// TwinCAT 3 PLC project Traffic
// ProgramVersion: 3.1.4024.0
// libraries:
//   Tc2_Standard, * (Beckhoff Automation GmbH)
//   Tc2_System, * (Beckhoff Automation GmbH)
//   Tc3_Module, * (Beckhoff Automation GmbH)
// project tree:
//   DUTs/ ST_ADJLIST.TcDUT, ST_ADJNODE.TcDUT, ST_GRAPH.TcDUT
//   GVLs/ CONSTANTS.TcGVL, GLOBALS.TcGVL
//   / PlcTask.TcTTO
//   POUs/ GET_MIN_DISTANCE_NODE.TcPOU, GET_SHORTEST_PATH.TcPOU, MAIN.TcPOU, DIJKSTRA.TcPOU, SIM_VALUES_CALC.TcPOU, TICK.TcPOU
// real-time tasks:
//   TASK PlcTask: cycle T#10ms, priority 20, ADS port 350

CONFIGURATION Traffic
    RESOURCE PLC ON TwinCAT3
        TASK PlcTask(INTERVAL := T#10ms, PRIORITY := 20);
        PROGRAM MAIN WITH PlcTask : MAIN;
    END_RESOURCE
END_CONFIGURATION

// ---- DUTs/ST_ADJLIST.TcDUT
TYPE ST_ADJLIST :
STRUCT
	aAdjNodes : ARRAY[1..3] OF POINTER TO ST_ADJNODE;
END_STRUCT
END_TYPE

// ---- DUTs/ST_ADJNODE.TcDUT
TYPE ST_ADJNODE :
STRUCT
	nNode	: INT;
	nWeight	: POINTER TO INT;
END_STRUCT
END_TYPE

// ---- DUTs/ST_GRAPH.TcDUT
TYPE ST_GRAPH :
STRUCT
	aAdjLists : ARRAY[1..24] OF POINTER TO ST_ADJLIST;
END_STRUCT
END_TYPE

// ---- GVLs/CONSTANTS.TcGVL
{attribute 'qualified_only'}
VAR_GLOBAL
	nIntMax : INT := 32767;
	
	// Base time in seconds required for <5 cars to pass through a crossroads.
	nBaseWeightSR : INT := 10;
	nBaseWeightL : INT := 20;
	
	// Most significant points in a made-up graph illustrating the intensity of traffic flow at specified hours.
	// aTrafficFlowTimes - X axis
	// aTrafficFlowVals - Y axis
	// To find the value of flow intensity inbetween these points, the following formula is used:
	// if (x2 < x1) x2 := x2 + 24; y := (x - x1) * (y2 - y1) / (x2 - x1) + y1;
	aTrafficFlowTimes : ARRAY[1..4] OF TOD := [TOD#4:0:0, TOD#9:0:0, TOD#12:0:0, TOD#17:0:0];
	aTrafficFlowVals : ARRAY[1..4] OF REAL := [0.0,       1.0,       0.5,        0.9];
	
	// Each day of the week has a different modifier for traffic intensity as well. 1 means Monday, 7 means Sunday.
	aTrafficFlowDaysVals : ARRAY[1..7] OF REAL := [1.0, 0.95, 0.9, 0.85, 0.8, 0.75, 0.7];
	
END_VAR

// ---- GVLs/GLOBALS.TcGVL
{attribute 'qualified_only'}
VAR_GLOBAL

// Settings for all crossroads.
// They indicate what number of cars should pass through specified parts of them when the modifier is 1.0.
// For example, setting nAHxSR to 100 on Mondays should result in 90 cars passing through at 17:00 and only 10 at 4:00.
// x - horizontal part
// y - vertical part
// SR - straights and rights
// L - lefts
nAHxSR, nAHySR, nAHxL, nAHyL : INT;
nBCxSR, nBCySR, nBCxL, nBCyL : INT;
nDExSR, nDEySR, nDExL, nDEyL : INT;
nFGxSR, nFGySR, nFGxL, nFGyL : INT;

// Depending on the time of day and day of week, this modifier will change from 0.0 for when there is no traffic to 1.0 at rush hours.
rModifier : REAL;

// Weights are the final product of nBaseWeightXX + nBaseWeightXX * {setting} / 5 * nModifier
// This is the time in seconds required to pass through a node.
nWeightAHxSR : INT;
nWeightAHySR : INT;
nWeightAHxL  : INT;
nWeightAHyL  : INT;

nWeightBCxSR : INT;
nWeightBCySR : INT;
nWeightBCxL  : INT;
nWeightBCyL  : INT;

nWeightDExSR : INT;
nWeightDEySR : INT;
nWeightDExL  : INT;
nWeightDEyL  : INT;

nWeightFGxSR : INT;
nWeightFGySR : INT;
nWeightFGxL  : INT;
nWeightFGyL  : INT;

// Adjacent nodes in adjacency lists. For example, stNode1to16 indicates the time required to get from node 1 to its adjacent node 16.
// ----- RIGHTS -----
//RIGHTS AH
stNode1to16  : ST_ADJNODE := (nNode:=16, nWeight:=ADR(nWeightAHySR));
stNode17to2  : ST_ADJNODE := (nNode:=2,  nWeight:=ADR(nWeightAHxSR));
stNode23to18 : ST_ADJNODE := (nNode:=18, nWeight:=ADR(nWeightAHySR));
stNode15to24 : ST_ADJNODE := (nNode:=24, nWeight:=ADR(nWeightAHxSR));
//RIGHTS BC
stNode3to17  : ST_ADJNODE := (nNode:=17, nWeight:=ADR(nWeightBCySR));
stNode5to4   : ST_ADJNODE := (nNode:=4,  nWeight:=ADR(nWeightBCxSR));
stNode20to6  : ST_ADJNODE := (nNode:=6,  nWeight:=ADR(nWeightBCySR));
stNode18to19 : ST_ADJNODE := (nNode:=19, nWeight:=ADR(nWeightBCxSR));
//RIGHTS DE
stNode19to21 : ST_ADJNODE := (nNode:=21, nWeight:=ADR(nWeightDEySR));
stNode7to20  : ST_ADJNODE := (nNode:=20, nWeight:=ADR(nWeightDExSR));
stNode9to8   : ST_ADJNODE := (nNode:=8,  nWeight:=ADR(nWeightDEySR));
stNode22to10 : ST_ADJNODE := (nNode:=10, nWeight:=ADR(nWeightDExSR));
//RIGHTS FG
stNode24to14 : ST_ADJNODE := (nNode:=14, nWeight:=ADR(nWeightFGySR));
stNode21to23 : ST_ADJNODE := (nNode:=23, nWeight:=ADR(nWeightFGxSR));
stNode11to22 : ST_ADJNODE := (nNode:=22, nWeight:=ADR(nWeightFGySR));
stNode13to12 : ST_ADJNODE := (nNode:=12, nWeight:=ADR(nWeightFGxSR));
// ----- STRAIGHTS -----
//STRAIGHTS AH
stNode1to24  : ST_ADJNODE := (nNode:=24, nWeight:=ADR(nWeightAHySR));
stNode23to2  : ST_ADJNODE := (nNode:=2,  nWeight:=ADR(nWeightAHySR));
stNode17to16 : ST_ADJNODE := (nNode:=16, nWeight:=ADR(nWeightAHxSR));
stNode15to18 : ST_ADJNODE := (nNode:=18, nWeight:=ADR(nWeightAHxSR));
//STRAIGHTS BC
stNode3to19 : ST_ADJNODE := (nNode:=19, nWeight:=ADR(nWeightBCySR));
stNode20to4 : ST_ADJNODE := (nNode:=4,  nWeight:=ADR(nWeightBCySR));
stNode5to17 : ST_ADJNODE := (nNode:=17, nWeight:=ADR(nWeightBCxSR));
stNode18to6 : ST_ADJNODE := (nNode:=6,  nWeight:=ADR(nWeightBCxSR));
//STRAIGHTS DE
stNode19to10 : ST_ADJNODE := (nNode:=10, nWeight:=ADR(nWeightDEySR));
stNode9to20  : ST_ADJNODE := (nNode:=20, nWeight:=ADR(nWeightDEySR));
stNode7to21  : ST_ADJNODE := (nNode:=21, nWeight:=ADR(nWeightDExSR));
stNode22to8  : ST_ADJNODE := (nNode:=8,  nWeight:=ADR(nWeightDExSR));
//STRAIGHTS FG
stNode24to12 : ST_ADJNODE := (nNode:=12, nWeight:=ADR(nWeightFGySR));
stNode11to23 : ST_ADJNODE := (nNode:=23, nWeight:=ADR(nWeightFGySR));
stNode21to14 : ST_ADJNODE := (nNode:=14, nWeight:=ADR(nWeightFGxSR));
stNode13to22 : ST_ADJNODE := (nNode:=22, nWeight:=ADR(nWeightFGxSR));
// ----- LEFTS -----
//LEFTS AH
stNode1to18  : ST_ADJNODE := (nNode:=18, nWeight:=ADR(nWeightAHyL));
stNode15to2  : ST_ADJNODE := (nNode:=2,  nWeight:=ADR(nWeightAHxL));
stNode17to24 : ST_ADJNODE := (nNode:=24, nWeight:=ADR(nWeightAHxL));
stNode23to16 : ST_ADJNODE := (nNode:=16, nWeight:=ADR(nWeightAHyL));
//LEFTS BC
stNode3to6   : ST_ADJNODE := (nNode:=6,  nWeight:=ADR(nWeightBCyL));
stNode18to4  : ST_ADJNODE := (nNode:=4,  nWeight:=ADR(nWeightBCxL));
stNode5to19  : ST_ADJNODE := (nNode:=19, nWeight:=ADR(nWeightBCxL));
stNode20to17 : ST_ADJNODE := (nNode:=17, nWeight:=ADR(nWeightBCyL));
//LEFTS DE
stNode19to8  : ST_ADJNODE := (nNode:=8,  nWeight:=ADR(nWeightDEyL));
stNode22to20 : ST_ADJNODE := (nNode:=20, nWeight:=ADR(nWeightDExL));
stNode7to10  : ST_ADJNODE := (nNode:=10, nWeight:=ADR(nWeightDExL));
stNode9to21  : ST_ADJNODE := (nNode:=21, nWeight:=ADR(nWeightDEyL));
//LEFTS FG
stNode24to22 : ST_ADJNODE := (nNode:=22, nWeight:=ADR(nWeightFGyL));
stNode13to23 : ST_ADJNODE := (nNode:=23, nWeight:=ADR(nWeightFGxL));
stNode21to12 : ST_ADJNODE := (nNode:=12, nWeight:=ADR(nWeightFGxL));
stNode11to14 : ST_ADJNODE := (nNode:=14, nWeight:=ADR(nWeightFGyL));

// Adjacency lists for all nodes that can act as sources. Note that there are no lists for destination-only nodes,
// namely nodes 2, 4, 6, 8, 10, 12, 14, 16.
stNodesFrom1  : ST_ADJLIST := (aAdjNodes:=[ADR(stNode1to16),  ADR(stNode1to18),  ADR(stNode1to24)]);
stNodesFrom3  : ST_ADJLIST := (aAdjNodes:=[ADR(stNode3to17),  ADR(stNode3to19),  ADR(stNode3to6)]);
stNodesFrom5  : ST_ADJLIST := (aAdjNodes:=[ADR(stNode5to17),  ADR(stNode5to19),  ADR(stNode5to4)]);
stNodesFrom7  : ST_ADJLIST := (aAdjNodes:=[ADR(stNode7to10),  ADR(stNode7to20),  ADR(stNode7to21)]);
stNodesFrom9  : ST_ADJLIST := (aAdjNodes:=[ADR(stNode9to20),  ADR(stNode9to21),  ADR(stNode9to8)]);
stNodesFrom11 : ST_ADJLIST := (aAdjNodes:=[ADR(stNode11to14), ADR(stNode11to22), ADR(stNode11to23)]);
stNodesFrom13 : ST_ADJLIST := (aAdjNodes:=[ADR(stNode13to12), ADR(stNode13to22), ADR(stNode13to23)]);
stNodesFrom15 : ST_ADJLIST := (aAdjNodes:=[ADR(stNode15to18), ADR(stNode15to2),  ADR(stNode15to24)]);
stNodesFrom17 : ST_ADJLIST := (aAdjNodes:=[ADR(stNode17to16), ADR(stNode17to2),  ADR(stNode17to24)]);
stNodesFrom18 : ST_ADJLIST := (aAdjNodes:=[ADR(stNode18to19), ADR(stNode18to4),  ADR(stNode18to6)]);
stNodesFrom19 : ST_ADJLIST := (aAdjNodes:=[ADR(stNode19to10), ADR(stNode19to21), ADR(stNode19to8)]);
stNodesFrom20 : ST_ADJLIST := (aAdjNodes:=[ADR(stNode20to17), ADR(stNode20to4),  ADR(stNode20to6)]);
stNodesFrom21 : ST_ADJLIST := (aAdjNodes:=[ADR(stNode21to12), ADR(stNode21to14), ADR(stNode21to23)]);
stNodesFrom22 : ST_ADJLIST := (aAdjNodes:=[ADR(stNode22to10), ADR(stNode22to20), ADR(stNode22to8)]);
stNodesFrom23 : ST_ADJLIST := (aAdjNodes:=[ADR(stNode23to16), ADR(stNode23to18), ADR(stNode23to2)]);
stNodesFrom24 : ST_ADJLIST := (aAdjNodes:=[ADR(stNode24to12), ADR(stNode24to14), ADR(stNode24to22)]);

// Adjacency graph. Note that destination-only nodes have no adjacency lists; their address is set to 0 and is ignored when searching.
stGraph : ST_GRAPH := (aAdjLists:=[
ADR(stNodesFrom1),
0,
ADR(stNodesFrom3),
0,
ADR(stNodesFrom5),
0,
ADR(stNodesFrom7),
0,
ADR(stNodesFrom9),
0,
ADR(stNodesFrom11),
0,
ADR(stNodesFrom13),
0,
ADR(stNodesFrom15),
0,
ADR(stNodesFrom17),
ADR(stNodesFrom18),
ADR(stNodesFrom19),
ADR(stNodesFrom20),
ADR(stNodesFrom21),
ADR(stNodesFrom22),
ADR(stNodesFrom23),
ADR(stNodesFrom24)]);

// Nodes for the Dijkstra algorithm search.
nStartPosition : INT := 1;
nEndPosition: INT := 2;

// List of all distances from nStartPosition
aDistances : ARRAY[1..24] OF INT;

// List of traveled nodes from nStartPosition to nEndPosition
aRoadFlags : ARRAY[1..24] OF BOOL;

END_VAR

// ---- POUs/MAIN.TcPOU
PROGRAM MAIN
VAR
	bShouldCalculate : BOOL;
END_VAR

TICK();
SIM_VALUES_CALC();
IF bShouldCalculate THEN
	DIJKSTRA();
	bShouldCalculate := FALSE;
END_IF

END_PROGRAM

// ---- POUs/TICK.TcPOU
PROGRAM TICK
VAR
	ins : BOOL;
	et : TIME;
	tick: TON;
	
	nDayOfTheWeek : INT := 1;
	
	tdSimTime : TOD := TOD#4:0:0;
	SimTime : UDINT;
	
	// Traffic flow time index for CONSTANTS.aTrafficFlowTimes
	x1i : INT := 1;
	x2i : INT := 2;
	x1, x2 : REAL;
	
	tdTickTime : TOD := TOD#0:15:0;
END_VAR
VAR // added by the converter: edge detectors and wires of the graphical bodies
    _w1, _w2, _w3 : BOOL;
END_VAR

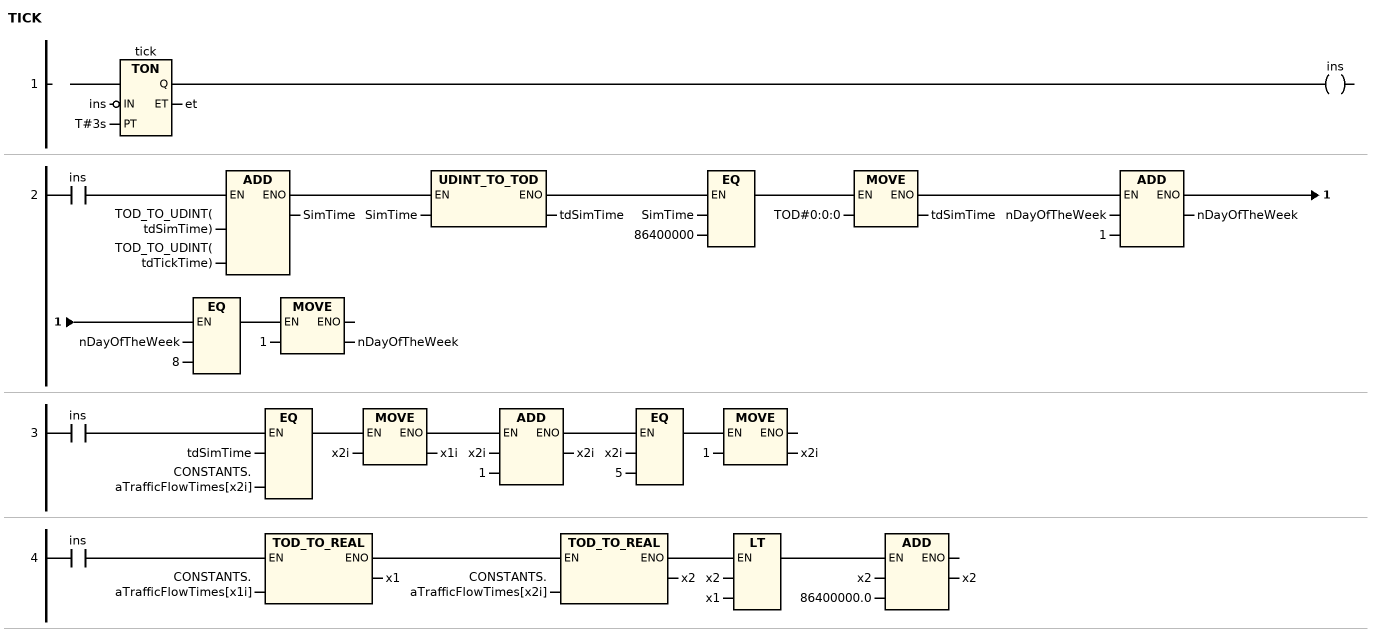
// NETWORK 1
tick(IN := NOT ins, PT := T#3s, ET => et); // TON
ins := tick.Q;

// NETWORK 2
_w1 := ins;
IF _w1 THEN SimTime := (TOD_TO_UDINT(tdSimTime)) + (TOD_TO_UDINT(tdTickTime)); END_IF
IF _w1 THEN tdSimTime := UDINT_TO_TOD(SimTime); END_IF
IF _w1 AND SimTime = 86400000 THEN tdSimTime := TOD#0:0:0; END_IF
IF _w1 AND SimTime = 86400000 THEN nDayOfTheWeek := nDayOfTheWeek + 1; END_IF
IF _w1 AND SimTime = 86400000 AND nDayOfTheWeek = 8 THEN nDayOfTheWeek := 1; END_IF

// NETWORK 3
_w2 := ins AND tdSimTime = CONSTANTS.aTrafficFlowTimes[x2i];
IF _w2 THEN x1i := x2i; END_IF
IF _w2 THEN x2i := x2i + 1; END_IF
IF _w2 AND x2i = 5 THEN x2i := 1; END_IF

// NETWORK 4
_w3 := ins;
IF _w3 THEN x1 := TOD_TO_REAL(CONSTANTS.aTrafficFlowTimes[x1i]); END_IF
IF _w3 THEN x2 := TOD_TO_REAL(CONSTANTS.aTrafficFlowTimes[x2i]); END_IF
IF _w3 AND x2 < x1 THEN x2 := x2 + 86400000.0; END_IF

END_PROGRAM

// ---- POUs/SIM_VALUES_CALC.TcPOU
PROGRAM SIM_VALUES_CALC
VAR
	x, x1, x2, y1, y2, y : REAL;	

	rPltMd: REAL;
	rPltMdL : REAL;
	rPltMdSR : REAL;
END_VAR

x := UDINT_TO_REAL(TICK.SimTime);

// TICK already does all the conversions and other necessary logic involving x1 and x2.
x1 := TICK.x1;
x2 := TICK.x2;

y1 := CONSTANTS.aTrafficFlowVals[TICK.x1i];
y2 := CONSTANTS.aTrafficFlowVals[TICK.x2i];

y := (y2 - y1) * (x - x1) / (x2 - x1) + y1;

GLOBALS.rModifier := y * CONSTANTS.aTrafficFlowDaysVals[TICK.nDayOfTheWeek];

rPltMd := 1.0 + GLOBALS.rModifier * 0.2;
rPltMdL := rPltMd * CONSTANTS.nBaseWeightL;
rPltMdSR := rPltMd * CONSTANTS.nBaseWeightSR;

GLOBALS.nWeightAHxL := REAL_TO_INT(GLOBALS.nAHxL * rPltMdL);
GLOBALS.nWeightAHyL := REAL_TO_INT(GLOBALS.nAHyL * rPltMdL);
GLOBALS.nWeightBCxL := REAL_TO_INT(GLOBALS.nBCxL * rPltMdL);
GLOBALS.nWeightBCyL := REAL_TO_INT(GLOBALS.nBCyL * rPltMdL);
GLOBALS.nWeightDExL := REAL_TO_INT(GLOBALS.nDExL * rPltMdL);
GLOBALS.nWeightDEyL := REAL_TO_INT(GLOBALS.nDEyL * rPltMdL);
GLOBALS.nWeightFGxL := REAL_TO_INT(GLOBALS.nFGxL * rPltMdL);
GLOBALS.nWeightFGyL := REAL_TO_INT(GLOBALS.nFGyL * rPltMdL);

GLOBALS.nWeightAHxSR := REAL_TO_INT(GLOBALS.nAHxSR * rPltMdL);
GLOBALS.nWeightAHySR := REAL_TO_INT(GLOBALS.nAHySR * rPltMdL);
GLOBALS.nWeightBCxSR := REAL_TO_INT(GLOBALS.nBCxSR * rPltMdL);
GLOBALS.nWeightBCySR := REAL_TO_INT(GLOBALS.nBCySR * rPltMdL);
GLOBALS.nWeightDExSR := REAL_TO_INT(GLOBALS.nDExSR * rPltMdL);
GLOBALS.nWeightDEySR := REAL_TO_INT(GLOBALS.nDEySR * rPltMdL);
GLOBALS.nWeightFGxSR := REAL_TO_INT(GLOBALS.nFGxSR * rPltMdL);
GLOBALS.nWeightFGySR := REAL_TO_INT(GLOBALS.nFGySR * rPltMdL);

END_PROGRAM

// ---- POUs/DIJKSTRA.TcPOU
FUNCTION DIJKSTRA
VAR
	i, nMinDistanceNode, nNodeInList, nAdjacentNode, nDistance: INT;
	aVisited : ARRAY[1..24] OF BOOL;
	aParents : ARRAY[1..24] OF INT;
END_VAR

FOR i := 1 TO 24 DO
	GLOBALS.aDistances[i] := CONSTANTS.nIntMax;
	GLOBALS.aRoadFlags[i] := FALSE;
END_FOR

GLOBALS.aDistances[GLOBALS.nStartPosition] := 0;

FOR i := 1 TO 24 DO
	nMinDistanceNode := GET_MIN_DISTANCE_NODE(GLOBALS.aDistances, aVisited);
	aVisited[nMinDistanceNode] := TRUE;
	
	IF NOT (GLOBALS.stGraph.aAdjLists[nMinDistanceNode] = 0) THEN
		FOR nNodeInList := 1 TO 3 DO
			nAdjacentNode := GLOBALS.stGraph.aAdjLists[nMinDistanceNode]^.aAdjNodes[nNodeInList]^.nNode;
			nDistance := GLOBALS.stGraph.aAdjLists[nMinDistanceNode]^.aAdjNodes[nNodeInList]^.nWeight^;
			// z tych 3 warunkow, warunek 2 chyba jest niepotrzebny ale nie pamietam
			IF NOT (aVisited[nAdjacentNode]) AND NOT (GLOBALS.aDistances[nMinDistanceNode] = CONSTANTS.nIntMax) AND (GLOBALS.aDistances[nMinDistanceNode] + nDistance < GLOBALS.aDistances[nAdjacentNode]) THEN
				GLOBALS.aDistances[nAdjacentNode] := GLOBALS.aDistances[nMinDistanceNode] + nDistance;
				aParents[nAdjacentNode] :=  nMinDistanceNode;
			END_IF
		END_FOR
	END_IF
END_FOR

GET_SHORTEST_PATH(GLOBALS.nEndPosition, aParents);

END_FUNCTION

// ---- POUs/GET_MIN_DISTANCE_NODE.TcPOU
FUNCTION GET_MIN_DISTANCE_NODE : INT
VAR_INPUT
	aDistances : ARRAY[1..24] OF INT;
	aVisited : ARRAY[1..24] OF BOOL;
END_VAR
VAR
	i, nMinIndex, nMinDistance : INT;
END_VAR

nMinIndex := -1;
nMinDistance := CONSTANTS.nIntMax;

FOR i := 1 TO 24 DO
	IF NOT (aVisited[i]) AND (aDistances[i] <= nMinDistance) THEN
		nMinDistance := aDistances[i];
		nMinIndex := i;
	END_IF
END_FOR

GET_MIN_DISTANCE_NODE := nMinIndex;

END_FUNCTION

// ---- POUs/GET_SHORTEST_PATH.TcPOU
FUNCTION GET_SHORTEST_PATH
VAR_INPUT
	nCurrentNode : INT;
	aParents : ARRAY[1..24] OF INT;
END_VAR
VAR
END_VAR

IF NOT (nCurrentNode = 0) THEN
	GET_SHORTEST_PATH(aParents[nCurrentNode], aParents);
	GLOBALS.aRoadFlags[nCurrentNode] := TRUE;
END_IF

END_FUNCTION
